{attribute 'GeneratedUsingTerminal: EK1122-0000-0018'}
{attribute addProperty BoxType "EK1122-0000-0018"}
{attribute addProperty Id "Beckhoff_EL3xxxsub_EK1100EK1100_1FC0878B2"}
{attribute addProperty CRC "3749281973"}
{attribute addProperty Size "2"}
TYPE Beckhoff_EL3xxxEK1122_DF7980B5 EXTENDS EK1122_1FC0878B :
STRUCT
	{attribute addProperty Name "Beckhoff_EL3xxxsub_EK1100"}
	{attribute addProperty PreviousPort "Beckhoff EL3xxxEK1122 : D"}
	Beckhoff_EL3xxxsub_EK1100 : EK1100_1FC0878B;
END_STRUCT
END_TYPE

(* stored: Version 1.2.0.0, ProductVersion 3.1.4024.9
   DUT Beckhoff_EL3xxxEK1122_DF7980B5: Id {b16af45a-38f2-4fe9-8d09-f9b4abfd189a} *)
